FUNCTION_BLOCK PartCount (* Basic Function Block Type *)
  (* Standard: 61499-2 *)
  (* Version 0.0, 2015-05-12, 4DIAC-IDE, 4DIAC-Consortium *)
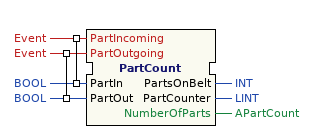
  EVENT_INPUT
    PartIncoming WITH PartIn; (* Confirms incoming part *)
    PartOutgoing WITH PartOut; (* Confirms outgoing part *)
  END_EVENT
  VAR_INPUT
    PartIn : BOOL; (* Sensor value for incoming parts *)
    PartOut : BOOL; (* Sensor value for outgoing parts *)
  END_VAR
  VAR_OUTPUT
    PartsOnBelt : INT;
    PartCounter : LINT;
  END_VAR
  PLUGS
    NumberOfParts : APartCount;
  END_PLUGS
  VAR
    lastIncrement : TIME; (* Internal Variable *)
    lastDecrement : TIME; (* Internal Variable *)
  END_VAR
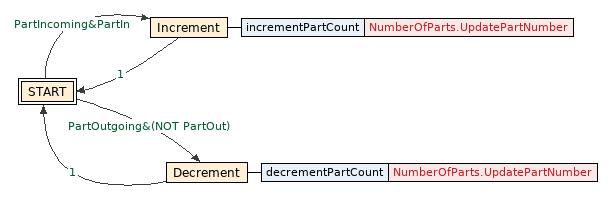
  EC_STATES
    START; (* Initial State *)
    Increment : incrementPartCount -> NumberOfParts.UpdatePartNumber; (* Initialization *)
    Decrement : decrementPartCount -> NumberOfParts.UpdatePartNumber; (* Normal execution *)
  END_STATES
  EC_TRANSITIONS
    START TO Increment := PartIncoming&PartIn;
    Increment TO START := 1;
    START TO Decrement := PartOutgoing&(NOT PartOut);
    Decrement TO START := 1;
  END_TRANSITIONS
  ALGORITHM incrementPartCount IN ST: (* increment number of parts on the belt *)
IF TIME() - lastIncrement > T#100ms THEN
  NumberOfParts.PartNumber := NumberOfParts.PartNumber + 1;
  PartCounter := PartCounter + 1;
END_IF;
PartsOnBelt := NumberOfParts.PartNumber;
lastIncrement := TIME();
  END_ALGORITHM
  ALGORITHM decrementPartCount IN ST: (* decrement number of parts on the belt *)
IF TIME() - lastDecrement  > T#100ms THEN
  NumberOfParts.PartNumber := NumberOfParts.PartNumber - 1;
END_IF;
PartsOnBelt := NumberOfParts.PartNumber;
lastIncrement := TIME();
  END_ALGORITHM
  SERVICE partCount_interface/partCount_implementation (* Basic Function Block Type *)
    SEQUENCE Increment
      partCount_interface.PartIncoming(PartIn = true) -> partCount_interface.NumberOfParts.UpdatePartNumber(PartsOnBelt = NumberOfParts.PartNumber; NumberOfParts.PartNumber>=; PartCounter>);
    END_SEQUENCE
    SEQUENCE Decrement
      partCount_interface.PartOutgoing(PartOut = false) -> partCount_interface.NumberOfParts.UpdatePartNumber(PartsOnBelt = NumberOfParts.PartNumber; NumberOfParts.PartNumber<=; PartCounter>=);
    END_SEQUENCE
  END_SERVICE
END_FUNCTION_BLOCK
